Fanuc KAREL source: kt00368.KL

-- PROVISIONAL review KL for V1013-1; original PC SHA256 3bf55748d2b410909e35e70718198f7609216812443618320a867a5dc79f8b9f
-- Incomplete behavior may be omitted. Consult companion uncertainty JSON. Do not deploy.
PROGRAM KT00368
%NOLOCKGROUP
VAR
  I1 : INTEGER
  OUT : BOOLEAN
-- UNRESOLVED_DECL H2 type=002017
BEGIN
  -- UNRESOLVED_PC offsets 5-16; opcodes 2E,23
  -- UNRESOLVED_PC offsets 21-35; opcodes 2E,22,9D,33,B4
  -- UNRESOLVED_PC offsets 40-62; opcodes 21,22,9D,33,B3,5A,23
  -- UNRESOLVED_PC offsets 67-71; opcodes 7F
END KT00368
